SUBAPPLICATION E_REND3 (* Subapplication Type *)
  (* Standard: 61499-2 *)
  (* Version 1.0, 2023-02-13, AK124017 *)
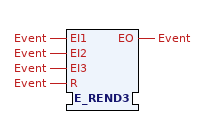
  EVENT_INPUT
    EI1;
    EI2;
    EI3;
    R;
  END_EVENT
  EVENT_OUTPUT
    EO;
  END_EVENT
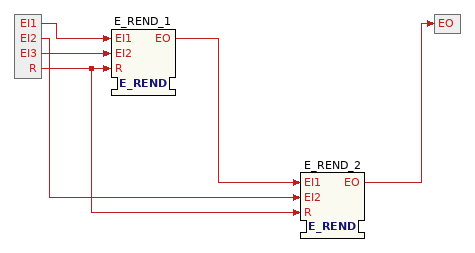
  FBS
    E_REND_1 : E_REND;
    E_REND_2 : E_REND;
  END_FBS
  EVENT_CONNECTIONS
    EI1 TO E_REND_1.EI1;
    EI2 TO E_REND_1.EI2;
    E_REND_1.EO TO E_REND_2.EI1;
    EI3 TO E_REND_2.EI2;
    R TO E_REND_1.R;
    R TO E_REND_2.R;
    E_REND_2.EO TO EO;
  END_CONNECTIONS
END_SUBAPPLICATION
